PROGRAM P_Demo_FB_HVAC2PointCtrl
VAR
    fb : FB_HVAC2PointCtrl;                            // 被演示 FB 实例
    eDataSecurityType_in : E_HVACDataSecurityType ;
    bSetDefault_in : BOOL := FALSE;
    bEnable_in : BOOL := FALSE;
    rW_in : REAL := 0.0;
    rX_in : REAL := 0.0;
    bReset_in : BOOL := FALSE;
    rHighLimit_io : REAL := 0.0;
    rLowLimit_io : REAL := 0.0;
    bDirection_io : BOOL := FALSE;
    tDelayOn_io : TIME := T#0S;
    tDelayOff_io : TIME := T#0S;
    bOut_out : BOOL;
    bInvalidParameter_out : BOOL;
END_VAR

// ============================================================================
// Tc2_HVAC.FB_HVAC2PointCtrl 演示程序
// ============================================================================
// 场景：把本 FB 实例化到一个 PLC 程序里，每周期单次调用；按需要把 VAR_INPUT 与
//       VAR_IN_OUT 接到工程信号；VAR_OUTPUT 写入对应监视变量。
// 价值：使用本 FB 比手写状态机 / 控制算法节省大量代码；与 Tc2_HVAC 体系内其它 FB
//       直接对接，命名 / 持久化 / 模式仲裁等约定一致。具体语义见 FB_HVAC2PointCtrl.md 主文档。
// 验证步骤：
//   1. 右键 PLC 项目下 POUs 文件夹 → Add → Existing Item → 选本 .TcPOU 文件
//   2. 引用 Tc2_HVAC（References → Add library）
//   3. 编译 → 登录 → 运行
//   4. 在线写各 *_in 输入信号触发 FB；在线 monitor *_out 引脚观察状态
// ============================================================================

fb(
    eDataSecurityType := eDataSecurityType_in,
    bSetDefault := bSetDefault_in,
    bEnable := bEnable_in,
    rW := rW_in,
    rX := rX_in,
    bReset := bReset_in,
    rHighLimit := rHighLimit_io,
    rLowLimit := rLowLimit_io,
    bDirection := bDirection_io,
    tDelayOn := tDelayOn_io,
    tDelayOff := tDelayOff_io,
    bOut => bOut_out,
    bInvalidParameter => bInvalidParameter_out
);

END_PROGRAM

(* stored: Version 1.1.0.1, ProductVersion 3.1.4024.5
   POU P_Demo_FB_HVAC2PointCtrl: Id {d8600cd7-7d98-5e0b-b4bd-3681a37b4b0a}, SpecialFunc None *)
